FUNCTION_BLOCK PhotoLumChuck EXTENDS ChuckBase
VAR_INPUT
	IoChuck : IoChuckPhotoLum;
END_VAR
VAR_OUTPUT
END_VAR
VAR
	{attribute 'OPC.UA.DA' := '0'}
	_config : PhotoLumChuckConfig;
	
	{attribute 'OPC.UA.DA' := '0'}
	_deliverMessages : INT;
	
	WaferPresenceMsg : STRING(255);
	
	{attribute 'OPC.UA.DA' := '0'}
	_initDevice : BOOL;
	
	{attribute 'OPC.UA.DA' := '0'}
	_itemInit : INT;
	
	{attribute 'OPC.UA.DA' := '0'}
	_itemScheduler : INT;
	{attribute 'OPC.UA.DA' := '0'}
	_itemRaisedProperties : INT;
	{attribute 'OPC.UA.DA' := '0'}
	_pulseGenerator : TON;
	
	{region 'Commands'}
		
	{attribute 'OPC.UA.DA' := '0'}			  		   
	_clampWaferCmd : BOOL;
	{attribute 'OPC.UA.DA' := '0'}			  		   
	_releaseWaferCmd : BOOL;
	{attribute 'OPC.UA.DA' := '0'}			  		   
	_raisePropertiesCmd : BOOL;
			
	{endregion}	
		
	{attribute 'OPC.UA.DA' := '0'}	
	_size : LREAL;	
		 
	{attribute 'OPC.UA.DA' := '0'}
	message : STRING;
	{attribute 'OPC.UA.DA' := '0'}
	_waferPresenceSensorCounter : UINT;			
	
	
	
END_VAR

SUPER^();

// Init device
InitDevice(); 

// Deliver messages
CASE _deliverMessages OF		
	EFeedbackMsgPhotoLumChuck.WaferPresenceMsg :
		WaferPresenceMsg := message;		
END_CASE
	
_deliverMessages := 0;

// Commands	
ClampWafer(_clampWaferCmd, _size);
ReleaseWafer(_releaseWaferCmd, _size);
RaisePropertiesChanged(_raisePropertiesCmd);

IF (NOT _raisePropertiesCmd) THEN
	MessageScheduler();
END_IF

{attribute 'TcRpcEnable' := '1'}
METHOD ClampWafer
VAR_INPUT
	Execute : BOOL;
	Value : LREAL;
END_VAR
VAR 
	size : EWaferSize := EWaferSize.Unknown;
END_VAR
IF Execute THEN
	_logger.Information(_message.Reset().Append(_config.Name).Append(' - Clamp wafer: ').Append(TO_STRING(Value)).ToString());

	CASE LREAL_TO_INT(Value) OF
		EWaferSize._100mm : 
			IoChuck.OutputVaccum100mm := TRUE;
			IoChuck.OutputVaccum150mm := FALSE; 
			IoChuck.OutputVaccum200mm := FALSE;			
			size := EWaferSize._100mm;
			
		EWaferSize._150mm :
			IoChuck.OutputVaccum100mm := FALSE;
			IoChuck.OutputVaccum150mm := TRUE; 
			IoChuck.OutputVaccum200mm := FALSE;
			size := EWaferSize._150mm;
			
		EWaferSize._200mm :
			IoChuck.OutputVaccum100mm := FALSE;
			IoChuck.OutputVaccum150mm := FALSE; 
			IoChuck.OutputVaccum200mm := TRUE;
			size := EWaferSize._200mm;
			
		EWaferSize.Unknown:		
			size := EWaferSize.Unknown;
			_logger.Warning(_message.Reset().Append(_config.Name).Append(' - Unknown size ').ToString());
	ELSE 
		_logger.Warning(_message.Reset().Append(_config.Name).Append(' - This size: ').Append(TO_STRING(Value)).Append(' does not exist').ToString());
	END_CASE
	
	WaferSize := size;
	
	_clampWaferCmd := FALSE;
END_IF
END_METHOD

METHOD FB_init : BOOL
VAR_INPUT
	bInitRetains : BOOL; // if TRUE, the retain variables are initialized (warm start / cold start)
	bInCopyCode : BOOL;  // if TRUE, the instance afterwards gets moved into the copy code (online change)
	Config : PhotoLumChuckConfig;
END_VAR
IF Config.IsEnabled THEN
	_config := Config;
	
	SUPER^._chuckConfig.Name := Config.Name;
	SUPER^._chuckConfig.DeviceID := Config.DeviceID;
	SUPER^._chuckConfig.IsEnabled := Config.IsEnabled;
	SUPER^._chuckConfig.LogLevel := Config.LogLevel;
	
	SUPER^.Name := Config.Name;
	SUPER^.DeviceID := Config.DeviceID;
	
	THIS^.Family := DeviceFamily.Chuck;

	THIS^.SetReady();
	_Logger.Information(_message.Reset().Append('Init ').
							Append('{').Append(TO_STRING(THIS^.Family)).Append('} - ').
							Append('{').Append(TO_STRING(THIS^.Name)).Append('} - ').
							Append('Status : ').Append(TO_STRING(THIS^.Status)).
							ToString());										 
END_IF
END_METHOD

METHOD InitDevice
VAR_INPUT
END_VAR
IF NOT _initDevice THEN			
	_logger.Information(_message.Reset().
								Append(_config.Name).
								Append(' - init device').ToString());		
								
	_initDevice := TRUE;
END_IF
END_METHOD

METHOD MessageScheduler
VAR_INPUT
END_VAR
IF _pulseGenerator.Q THEN
	_pulseGenerator(IN := FALSE, PT := T#10MS);
		
	CASE _itemScheduler OF	
		0:	WaferPresenceMsg := ' ';
			_itemScheduler := 1;
	
		1:	ReadWaferPresence();
			_itemScheduler := 0;		
									
	END_CASE
ELSE
	_pulseGenerator(IN := TRUE, PT := T#100MS);	
END_IF
END_METHOD

{attribute 'TcRpcEnable' := '1'}
METHOD RaisePropertiesChanged
VAR_INPUT
	Execute : BOOL;
END_VAR
IF Execute THEN		
	_raisePropertiesCmd := TRUE;	
	
	IF _pulseGenerator.Q THEN
		_pulseGenerator(IN := FALSE, PT := T#10MS);
		
		CASE _itemRaisedProperties OF		
			0: _itemRaisedProperties := 10;
				
			10: _logger.Information(_message.Reset().Append(_config.Name).Append(' - RaisePropertiesChanged').ToString());
				_raisePropertiesCmd := FALSE;
				_itemRaisedProperties := 0;		
		END_CASE	
	ELSE
		_pulseGenerator(IN := TRUE, PT := T#100MS);	
	END_IF		
END_IF
END_METHOD

METHOD ReadWaferPresence
VAR_INPUT
END_VAR
VAR	
	waferPresence : STRING;
	diameter : STRING;
END_VAR
_deliverMessages := EFeedbackMsgPsdChuck.WaferPresenceMsg;

IF _waferPresenceSensorCounter < Const.PHOTOLUM_NUMBER_WAFER_PRESENCE_SENSORS - 1 THEN
	_waferPresenceSensorCounter := _waferPresenceSensorCounter + 1;
ELSE
	_waferPresenceSensorCounter := 0;
END_IF

diameter := TO_STRING(_config.WaferPresenceSensor[_waferPresenceSensorCounter].Diameter);

IF _config.WaferPresenceSensor[_waferPresenceSensorCounter].InputWaferPresence AND 
   _config.WaferPresenceSensor[_waferPresenceSensorCounter].Diameter = TO_UINT(_waferSize) THEN
	waferPresence := INT_TO_STRING(EMaterialPresence.Present);
ELSE
	waferPresence := INT_TO_STRING(EMaterialPresence.NotPresent);		
END_IF

message := CONCAT(CONCAT(diameter, ';'), waferPresence);
END_METHOD

{attribute 'TcRpcEnable' := '1'}
METHOD ReleaseWafer
VAR_INPUT
	Execute : BOOL;
	Value : LREAL;
END_VAR
IF Execute THEN
	_logger.Information(_message.Reset().Append(_config.Name).Append(' - release wafer: ').Append(TO_STRING(Value)).ToString());

	IF Value = EWaferSize._100mm THEN
		IoChuck.OutputVaccum100mm := FALSE;
	ELSIF Value = EWaferSize._150mm THEN		
		IoChuck.OutputVaccum150mm := FALSE; 		
	ELSIF Value = EWaferSize._200mm THEN
		IoChuck.OutputVaccum200mm := FALSE;
	ELSIF Value = EWaferSize.Unknown THEN
		_logger.Warning(_message.Reset().Append(_config.Name).Append(' - Unknown size ').ToString());
	ELSE 
		_logger.Warning(_message.Reset().Append(_config.Name).Append(' - This size: ').Append(TO_STRING(Value)).Append(' does not exist').ToString());
	END_IF

	WaferSize := EWaferSize.Unknown;
	
	_releaseWaferCmd := FALSE;
END_IF
END_METHOD

END_FUNCTION_BLOCK

(* stored: Version 1.1.0.1, ProductVersion 3.1.4024.12
   POU PhotoLumChuck: Id {4a95dd5a-ee7c-4712-abd8-2388e2a4165b}, SpecialFunc None
   Folder Commands: Id {a97a6e70-5f2e-4ff9-9af5-ee69a5038400}
   Method ClampWafer: Id {3e46cccb-4e8e-4d04-b108-54a6a8830e24}
   Method FB_init: Id {c6c17ee1-7725-4610-be5f-46a553ac8095}
   Method InitDevice: Id {e851f87d-d091-4527-a40f-c2bee8cd0dc7}
   Method MessageScheduler: Id {e0d7da2c-466c-4a66-bee4-bfcec3f15fc0}
   Method RaisePropertiesChanged: Id {30b5bf2f-d4af-4fcf-82bf-553fd8f4f061}
   Method ReadWaferPresence: Id {f9626d81-8d28-4763-81a1-924a18920772}
   Method ReleaseWafer: Id {b19b51df-5643-43e4-a0aa-4c532361b6ea} *)
